{attribute 'GeneratedUsingTerminal: EL3152--0000'}
{attribute addProperty BoxType "EL3152--0000"}
{attribute addProperty Description "EL3152 2Ch. Ana. Input 4-20mA"}
{attribute addProperty Physics "KK"}
{attribute addProperty Id "Channel_1AT %I*Channel_7539AA333Channel_2AT %I*Channel_7539AA333WcStateAT %I*WcState_9091E0EB2InfoDataAT %I*InfoData_32EB74EA10"}
{attribute addProperty CRC "2161773851"}
{attribute addProperty Size "18"}
TYPE EL3152_80DA0D1B EXTENDS EtcSlaveTerminalBase_947E5A46 :
STRUCT
	{attribute addProperty Name "Channel_1"}
	Channel_1 : Channel_7539AA33;
	{attribute addProperty Name "Channel_2"}
	Channel_2 : Channel_7539AA33;
	{attribute addProperty Name "WcState"}
	WcState : WcState_9091E0EB;
	{attribute addProperty Name "InfoData"}
	InfoData : InfoData_32EB74EA;
END_STRUCT
END_TYPE

(* stored: Version 1.2.0.0, ProductVersion 3.1.4024.11
   DUT EL3152_80DA0D1B: Id {2a1e2267-e113-4dd3-9b3a-a88c3bedc239} *)
